(* 
| :Description: This function block represents basic digital input and can be used for creating an instance of signle digital input device like buttons, switches, sensors.
| To get the current status of digital input use "Value" property. To simulate state of the input by software set "Enable Force" parameter and change value via "MR_ResetForceValue" and "MR_SetForceValue" methods.
*)
FUNCTION_BLOCK FB_DigitalInput EXTENDS FB_DigitalDevice IMPLEMENTS I_DigitalInput
VAR
	(* Internal status *)
	bIn				AT %I*	: BOOL;		(* Current value of input *)
	bInForced				: BOOL;		(* Forced value from software *)
	bEnableForce			: BOOL;		(* Enable forcing of the input from software *)
	bRisingTrigger 			: BOOL;		(* Rising trigger of input detected*)
	bFallingTrigger 		: BOOL;		(* Falling trigger of input detected*)
	
	(* Function blocks *)
	rtRisingTrigger 		: R_TRIG;	(* Rising trigger detecting FB*)
	ftFallingTrigger		: F_TRIG;	(* Falling trigger detecting FB*)
END_VAR

PROPERTY EnableForce : BOOL
GET
EnableForce := bEnableForce;
END_GET
SET
bEnableForce := EnableForce;
END_SET
END_PROPERTY

PROPERTY FallingTrigger : BOOL
GET
ftFallingTrigger(CLK := In, Q => bFallingTrigger);
FallingTrigger := bFallingTrigger;
END_GET
END_PROPERTY

PROPERTY In : BOOL
GET
IF NOT bEnableForce THEN
	In := bIn;
ELSE
	In := bInForced;
END_IF
END_GET
END_PROPERTY

METHOD MR_ResetForceValue
IF bEnableForce THEN
	bInForced := FALSE;
	
END_IF
END_METHOD

METHOD MR_SetForceValue
IF bEnableForce THEN
	bInForced := TRUE;
	
END_IF
END_METHOD

PROPERTY RisingTrigger : BOOL
GET
rtRisingTrigger(CLK := In, Q => bRisingTrigger);
RisingTrigger := bRisingTrigger;
END_GET
END_PROPERTY

END_FUNCTION_BLOCK

(* stored: Version 1.1.0.1, ProductVersion 3.1.4024.12
   POU FB_DigitalInput: Id {bedeeace-128a-4c52-a09e-68eee13bdaca}, SpecialFunc None
   Folder Properties: Id {b9c448b3-015a-44fc-9825-650c8552021d}
   Folder Parameters: Id {62c40e2f-6a2c-4616-9168-b453c85c815f}
   Folder Status: Id {9d3f748c-cf49-4e67-bfe7-a00e3a535781}
   Folder Requests: Id {ac88b929-e11a-4b07-bd28-9602c1ffbbea}
   Property EnableForce: Id {bdfe49aa-0cd9-495a-bfe3-ba0f2883f93c}
   Get Get: Id {6022955a-088a-4b51-99f2-296c5d1da40e}
   Set Set: Id {5f2cee22-a1ed-4d67-9b66-d992c03f92bb}
   Property FallingTrigger: Id {89ab6be1-df5f-4135-99f6-4f2830efe301}
   Get Get: Id {91c4fbc0-f0d6-4b90-81fe-93c958d6a12d}
   Property In: Id {38e6612d-c4f4-4e0f-a4ea-d83d9f98eecd}
   Get Get: Id {559f91e4-b94e-4738-9826-22c596939736}
   Method MR_ResetForceValue: Id {e2b4a578-5d65-4952-82bd-2175d9340fb3}
   Method MR_SetForceValue: Id {79c40443-22cb-40ff-a385-3d72febf89e3}
   Property RisingTrigger: Id {e110483b-491c-42f8-99ac-6a8177cd245c}
   Get Get: Id {4725f269-654a-44da-9533-fda36787b607} *)
